// TIA Portal V16 export
// export: Created 2021-10-20T17:33:50.8567444Z, ExportSetting WithDefaults, DisplayName Totally Integrated Automation Portal, DisplayVersion V16, DisplayName TIA Portal Version Control Interface, DisplayVersion V16, DisplayName TIA Portal Openness, DisplayVersion V16, DisplayName TIA Portal Teamcenter Gateway, DisplayVersion V16, DisplayName SINAMICS Startdrive Advanced, DisplayVersion V16, DisplayName SINAMICS Startdrive G130, G150, S120, S150, SINAMICS MV, S210, DisplayVersion V16, DisplayName SINAMICS Startdrive G110M, G120, G120C, G120D, G120P, DisplayVersion V16, DisplayName STEP 7 Professional, DisplayVersion V16, DisplayName STEP 7 Safety, DisplayVersion V16, DisplayName WinCC Advanced, DisplayVersion V16
FUNCTION_BLOCK "Chillgard"   // FB2, LAD
TITLE = Chillgard analog communications
{ S7_Optimized_Access := 'TRUE' }
VERSION : 0.1
// Currently the Chillgard is only sensing 410A refrigerant.  More gas profiles may be added later.
// 
// Chillgard 5000 measures Rooms 16 & 19 - Indoor room, Indoor unit, Outdoor room, and Outdoor unit
// stored: AutoNumber true, IsIECCheckEnabled false, IsRetainMemResEnabled false, MemoryReserve 100, SetENOAutomatically false, UDAEnableTagReadback false
   VAR_TEMP   // added for the SCL form of the ladder/FBD networks
      _w1 : Bool;
      _w2 : Bool;
      _w3 : Bool;
      _w4 : Bool;
   END_VAR
BEGIN

REGION Network 1: Read and scale analog input values
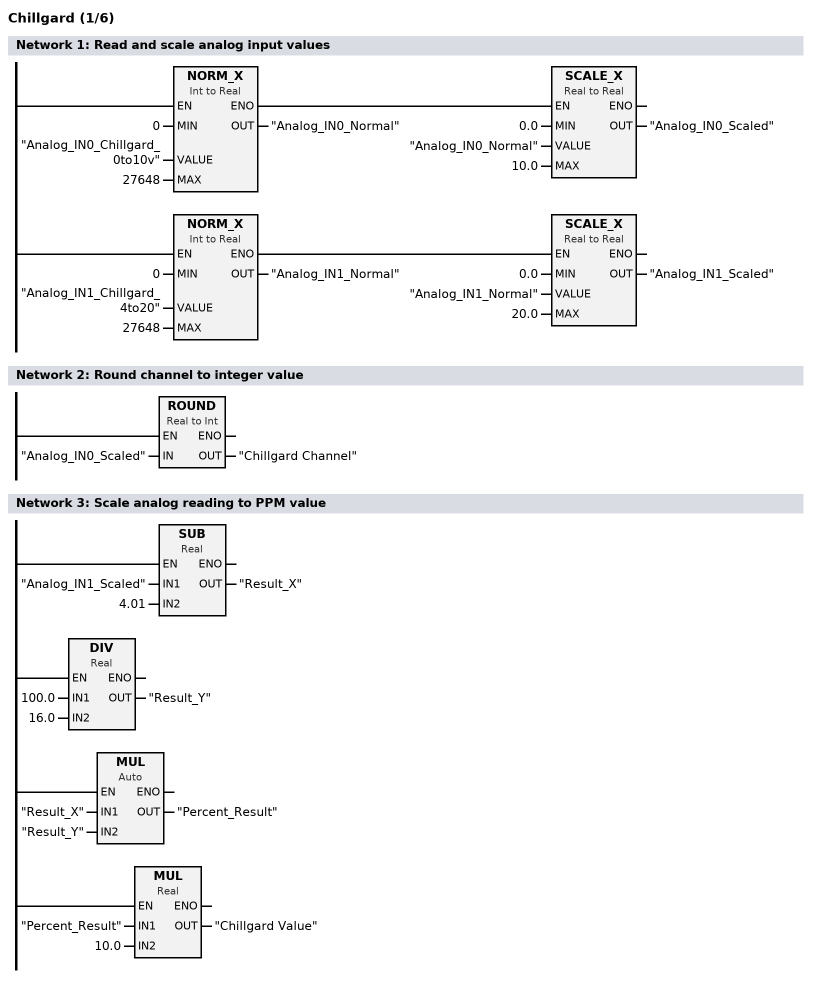
   RUNG wire#powerrail
      { S7_Templates := "[SrcType := Int, DestType := Real]" } Normalize(min := 0, value := "Analog_IN0_Chillgard_0to10v", max := 27648, out => "Analog_IN0_Normal")
      { S7_Templates := "[SrcType := Real, DestType := Real]" } Scale(min := 0.0, value := "Analog_IN0_Normal", max := 10.0, out => "Analog_IN0_Scaled")
   END_RUNG
   RUNG wire#powerrail
      { S7_Templates := "[SrcType := Int, DestType := Real]" } Normalize(min := 0, value := "Analog_IN1_Chillgard_4to20", max := 27648, out => "Analog_IN1_Normal")
      { S7_Templates := "[SrcType := Real, DestType := Real]" } Scale(min := 0.0, value := "Analog_IN1_Normal", max := 20.0, out => "Analog_IN1_Scaled")
   END_RUNG
   // the same network as SCL:
   "Analog_IN0_Normal" := NORM_X(MIN := 0, VALUE := "Analog_IN0_Chillgard_0to10v", MAX := 27648);
   "Analog_IN0_Scaled" := SCALE_X(MIN := 0.0, VALUE := "Analog_IN0_Normal", MAX := 10.0);
   "Analog_IN1_Normal" := NORM_X(MIN := 0, VALUE := "Analog_IN1_Chillgard_4to20", MAX := 27648);
   "Analog_IN1_Scaled" := SCALE_X(MIN := 0.0, VALUE := "Analog_IN1_Normal", MAX := 20.0);
END_REGION

REGION Network 2: Round channel to integer value
   RUNG wire#powerrail
      { S7_Templates := "[SrcType := Real, DestType := Int]" } Round(in := "Analog_IN0_Scaled", out => "Chillgard Channel")
   END_RUNG
   // the same network as SCL:
   "Chillgard Channel" := ROUND("Analog_IN0_Scaled");
END_REGION

REGION Network 3: Scale analog reading to PPM value
   RUNG wire#powerrail
      { S7_Templates := "SrcType := Real" } Sub(in1 := "Analog_IN1_Scaled", in2 := 4.01, out => "Result_X")
   END_RUNG
   RUNG wire#powerrail
      { S7_Templates := "SrcType := Real" } Div(in1 := 100.0, in2 := 16.0, out => "Result_Y")
   END_RUNG
   RUNG wire#powerrail
      Mul(in1 := "Result_X", in2 := "Result_Y", out => "Percent_Result")
   END_RUNG
   RUNG wire#powerrail
      { S7_Templates := "SrcType := Real" } Mul(in1 := "Percent_Result", in2 := 10.0, out => "Chillgard Value")
   END_RUNG
   // the same network as SCL:
   "Result_X" := "Analog_IN1_Scaled" - 4.01;
   "Result_Y" := 100.0 / 16.0;
   "Percent_Result" := "Result_X" * "Result_Y";
   "Chillgard Value" := "Percent_Result" * 10.0;
END_REGION

REGION Network 4: Assign values to proper channels - Room 4
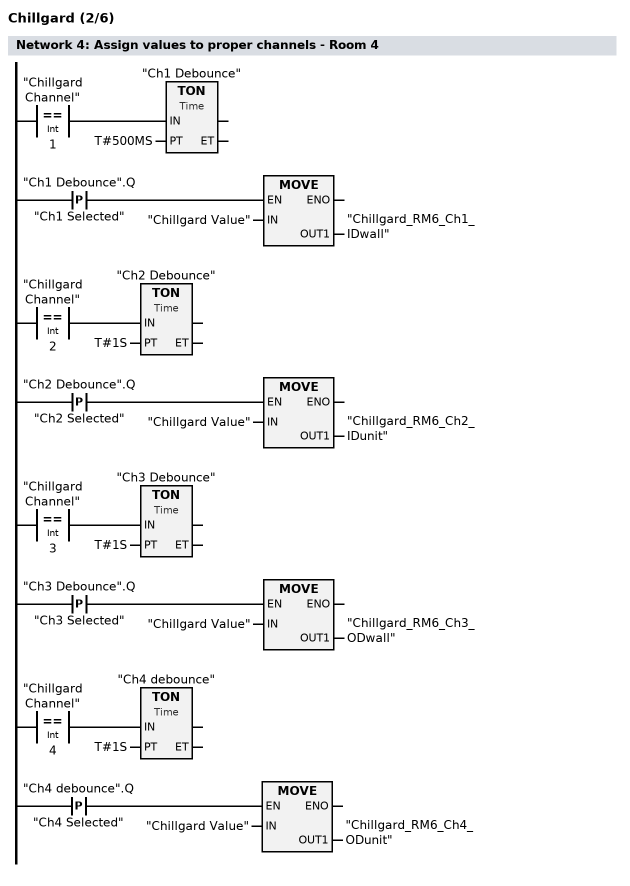
   RUNG wire#powerrail
      { S7_Templates := "SrcType := Int" } EQ_Contact(in1 := "Chillgard Channel", in2 := 1)
      { S7_Templates := "time_type := Time" } "Ch1 Debounce".TON(pt := T#500MS, et =>)
   END_RUNG
   RUNG wire#powerrail
      P_Contact(operand := "Ch1 Debounce".Q, bit := "Ch1 Selected")
      Move(in := "Chillgard Value", out1 => "Chillgard_RM6_Ch1_IDwall")
   END_RUNG
   RUNG wire#powerrail
      { S7_Templates := "SrcType := Int" } EQ_Contact(in1 := "Chillgard Channel", in2 := 2)
      { S7_Templates := "time_type := Time" } "Ch2 Debounce".TON(pt := T#1S, et =>)
   END_RUNG
   RUNG wire#powerrail
      P_Contact(operand := "Ch2 Debounce".Q, bit := "Ch2 Selected")
      Move(in := "Chillgard Value", out1 => "Chillgard_RM6_Ch2_IDunit")
   END_RUNG
   RUNG wire#powerrail
      { S7_Templates := "SrcType := Int" } EQ_Contact(in1 := "Chillgard Channel", in2 := 3)
      { S7_Templates := "time_type := Time" } "Ch3 Debounce".TON(pt := T#1S, et =>)
   END_RUNG
   RUNG wire#powerrail
      P_Contact(operand := "Ch3 Debounce".Q, bit := "Ch3 Selected")
      Move(in := "Chillgard Value", out1 => "Chillgard_RM6_Ch3_ODwall")
   END_RUNG
   RUNG wire#powerrail
      { S7_Templates := "SrcType := Int" } EQ_Contact(in1 := "Chillgard Channel", in2 := 4)
      { S7_Templates := "time_type := Time" } "Ch4 debounce".TON(pt := T#1S, et =>)
   END_RUNG
   RUNG wire#powerrail
      P_Contact(operand := "Ch4 debounce".Q, bit := "Ch4 Selected")
      Move(in := "Chillgard Value", out1 => "Chillgard_RM6_Ch4_ODunit")
   END_RUNG
   // the same network as SCL:
   "Ch1 Debounce".TON(IN := "Chillgard Channel" = 1, PT := T#500MS);
   #_w1 := "Ch1 Debounce".Q AND NOT "Ch1 Selected";   // rising edge of "Ch1 Debounce".Q
   "Ch1 Selected" := "Ch1 Debounce".Q;
   IF #_w1 THEN "Chillgard_RM6_Ch1_IDwall" := "Chillgard Value"; END_IF;
   "Ch2 Debounce".TON(IN := "Chillgard Channel" = 2, PT := T#1S);
   #_w2 := "Ch2 Debounce".Q AND NOT "Ch2 Selected";   // rising edge of "Ch2 Debounce".Q
   "Ch2 Selected" := "Ch2 Debounce".Q;
   IF #_w2 THEN "Chillgard_RM6_Ch2_IDunit" := "Chillgard Value"; END_IF;
   "Ch3 Debounce".TON(IN := "Chillgard Channel" = 3, PT := T#1S);
   #_w3 := "Ch3 Debounce".Q AND NOT "Ch3 Selected";   // rising edge of "Ch3 Debounce".Q
   "Ch3 Selected" := "Ch3 Debounce".Q;
   IF #_w3 THEN "Chillgard_RM6_Ch3_ODwall" := "Chillgard Value"; END_IF;
   "Ch4 debounce".TON(IN := "Chillgard Channel" = 4, PT := T#1S);
   #_w4 := "Ch4 debounce".Q AND NOT "Ch4 Selected";   // rising edge of "Ch4 debounce".Q
   "Ch4 Selected" := "Ch4 debounce".Q;
   IF #_w4 THEN "Chillgard_RM6_Ch4_ODunit" := "Chillgard Value"; END_IF;
END_REGION

REGION Network 5: Assign values to proper channels - Room 5
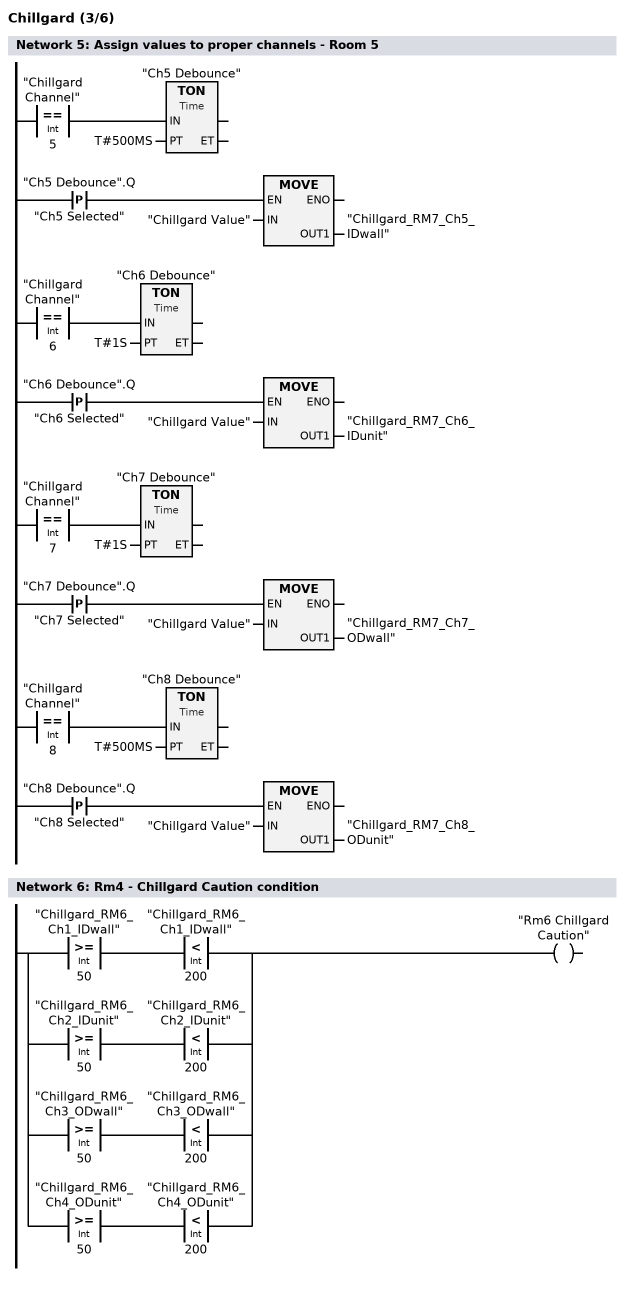
   RUNG wire#powerrail
      { S7_Templates := "SrcType := Int" } EQ_Contact(in1 := "Chillgard Channel", in2 := 5)
      { S7_Templates := "time_type := Time" } "Ch5 Debounce".TON(pt := T#500MS, et =>)
   END_RUNG
   RUNG wire#powerrail
      P_Contact(operand := "Ch5 Debounce".Q, bit := "Ch5 Selected")
      Move(in := "Chillgard Value", out1 => "Chillgard_RM7_Ch5_IDwall")
   END_RUNG
   RUNG wire#powerrail
      { S7_Templates := "SrcType := Int" } EQ_Contact(in1 := "Chillgard Channel", in2 := 6)
      { S7_Templates := "time_type := Time" } "Ch6 Debounce".TON(pt := T#1S, et =>)
   END_RUNG
   RUNG wire#powerrail
      P_Contact(operand := "Ch6 Debounce".Q, bit := "Ch6 Selected")
      Move(in := "Chillgard Value", out1 => "Chillgard_RM7_Ch6_IDunit")
   END_RUNG
   RUNG wire#powerrail
      { S7_Templates := "SrcType := Int" } EQ_Contact(in1 := "Chillgard Channel", in2 := 7)
      { S7_Templates := "time_type := Time" } "Ch7 Debounce".TON(pt := T#1S, et =>)
   END_RUNG
   RUNG wire#powerrail
      P_Contact(operand := "Ch7 Debounce".Q, bit := "Ch7 Selected")
      Move(in := "Chillgard Value", out1 => "Chillgard_RM7_Ch7_ODwall")
   END_RUNG
   RUNG wire#powerrail
      { S7_Templates := "SrcType := Int" } EQ_Contact(in1 := "Chillgard Channel", in2 := 8)
      { S7_Templates := "time_type := Time" } "Ch8 Debounce".TON(pt := T#500MS, et =>)
   END_RUNG
   RUNG wire#powerrail
      P_Contact(operand := "Ch8 Debounce".Q, bit := "Ch8 Selected")
      Move(in := "Chillgard Value", out1 => "Chillgard_RM7_Ch8_ODunit")
   END_RUNG
   // the same network as SCL:
   "Ch5 Debounce".TON(IN := "Chillgard Channel" = 5, PT := T#500MS);
   #_w1 := "Ch5 Debounce".Q AND NOT "Ch5 Selected";   // rising edge of "Ch5 Debounce".Q
   "Ch5 Selected" := "Ch5 Debounce".Q;
   IF #_w1 THEN "Chillgard_RM7_Ch5_IDwall" := "Chillgard Value"; END_IF;
   "Ch6 Debounce".TON(IN := "Chillgard Channel" = 6, PT := T#1S);
   #_w2 := "Ch6 Debounce".Q AND NOT "Ch6 Selected";   // rising edge of "Ch6 Debounce".Q
   "Ch6 Selected" := "Ch6 Debounce".Q;
   IF #_w2 THEN "Chillgard_RM7_Ch6_IDunit" := "Chillgard Value"; END_IF;
   "Ch7 Debounce".TON(IN := "Chillgard Channel" = 7, PT := T#1S);
   #_w3 := "Ch7 Debounce".Q AND NOT "Ch7 Selected";   // rising edge of "Ch7 Debounce".Q
   "Ch7 Selected" := "Ch7 Debounce".Q;
   IF #_w3 THEN "Chillgard_RM7_Ch7_ODwall" := "Chillgard Value"; END_IF;
   "Ch8 Debounce".TON(IN := "Chillgard Channel" = 8, PT := T#500MS);
   #_w4 := "Ch8 Debounce".Q AND NOT "Ch8 Selected";   // rising edge of "Ch8 Debounce".Q
   "Ch8 Selected" := "Ch8 Debounce".Q;
   IF #_w4 THEN "Chillgard_RM7_Ch8_ODunit" := "Chillgard Value"; END_IF;
END_REGION

REGION Network 6: Rm4 - Chillgard Caution condition
   RUNG wire#powerrail
      { S7_Templates := "SrcType := Int" } GE_Contact(in1 := "Chillgard_RM6_Ch1_IDwall", in2 := 50)
      { S7_Templates := "SrcType := Int" } LT_Contact(in1 := "Chillgard_RM6_Ch1_IDwall", in2 := 200)
      wire#w1
      Coil( "Rm6 Chillgard Caution" )
   END_RUNG
   RUNG wire#powerrail
      { S7_Templates := "SrcType := Int" } GE_Contact(in1 := "Chillgard_RM6_Ch2_IDunit", in2 := 50)
      { S7_Templates := "SrcType := Int" } LT_Contact(in1 := "Chillgard_RM6_Ch2_IDunit", in2 := 200)
   END_RUNG wire#w1
   RUNG wire#powerrail
      { S7_Templates := "SrcType := Int" } GE_Contact(in1 := "Chillgard_RM6_Ch3_ODwall", in2 := 50)
      { S7_Templates := "SrcType := Int" } LT_Contact(in1 := "Chillgard_RM6_Ch3_ODwall", in2 := 200)
   END_RUNG wire#w1
   RUNG wire#powerrail
      { S7_Templates := "SrcType := Int" } GE_Contact(in1 := "Chillgard_RM6_Ch4_ODunit", in2 := 50)
      { S7_Templates := "SrcType := Int" } LT_Contact(in1 := "Chillgard_RM6_Ch4_ODunit", in2 := 200)
   END_RUNG wire#w1
   // the same network as SCL:
   "Rm6 Chillgard Caution" := (("Chillgard_RM6_Ch1_IDwall" >= 50) AND ("Chillgard_RM6_Ch1_IDwall" < 200)) OR (("Chillgard_RM6_Ch2_IDunit" >= 50) AND ("Chillgard_RM6_Ch2_IDunit" < 200)) OR (("Chillgard_RM6_Ch3_ODwall" >= 50) AND ("Chillgard_RM6_Ch3_ODwall" < 200)) OR (("Chillgard_RM6_Ch4_ODunit" >= 50) AND ("Chillgard_RM6_Ch4_ODunit" < 200));
END_REGION

REGION Network 7: Rm4 - Chillgard Warning Condition
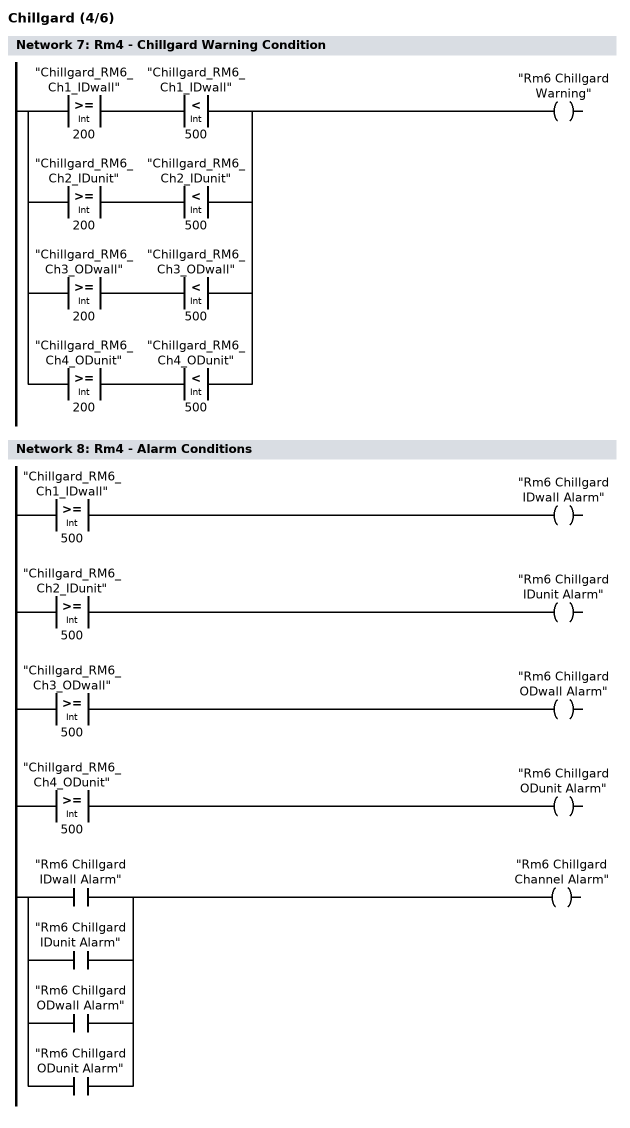
   RUNG wire#powerrail
      { S7_Templates := "SrcType := Int" } GE_Contact(in1 := "Chillgard_RM6_Ch1_IDwall", in2 := 200)
      { S7_Templates := "SrcType := Int" } LT_Contact(in1 := "Chillgard_RM6_Ch1_IDwall", in2 := 500)
      wire#w1
      Coil( "Rm6 Chillgard Warning" )
   END_RUNG
   RUNG wire#powerrail
      { S7_Templates := "SrcType := Int" } GE_Contact(in1 := "Chillgard_RM6_Ch2_IDunit", in2 := 200)
      { S7_Templates := "SrcType := Int" } LT_Contact(in1 := "Chillgard_RM6_Ch2_IDunit", in2 := 500)
   END_RUNG wire#w1
   RUNG wire#powerrail
      { S7_Templates := "SrcType := Int" } GE_Contact(in1 := "Chillgard_RM6_Ch3_ODwall", in2 := 200)
      { S7_Templates := "SrcType := Int" } LT_Contact(in1 := "Chillgard_RM6_Ch3_ODwall", in2 := 500)
   END_RUNG wire#w1
   RUNG wire#powerrail
      { S7_Templates := "SrcType := Int" } GE_Contact(in1 := "Chillgard_RM6_Ch4_ODunit", in2 := 200)
      { S7_Templates := "SrcType := Int" } LT_Contact(in1 := "Chillgard_RM6_Ch4_ODunit", in2 := 500)
   END_RUNG wire#w1
   // the same network as SCL:
   "Rm6 Chillgard Warning" := (("Chillgard_RM6_Ch1_IDwall" >= 200) AND ("Chillgard_RM6_Ch1_IDwall" < 500)) OR (("Chillgard_RM6_Ch2_IDunit" >= 200) AND ("Chillgard_RM6_Ch2_IDunit" < 500)) OR (("Chillgard_RM6_Ch3_ODwall" >= 200) AND ("Chillgard_RM6_Ch3_ODwall" < 500)) OR (("Chillgard_RM6_Ch4_ODunit" >= 200) AND ("Chillgard_RM6_Ch4_ODunit" < 500));
END_REGION

REGION Network 8: Rm4 - Alarm Conditions
   RUNG wire#powerrail
      { S7_Templates := "SrcType := Int" } GE_Contact(in1 := "Chillgard_RM6_Ch1_IDwall", in2 := 500)
      Coil( "Rm6 Chillgard IDwall Alarm" )
   END_RUNG
   RUNG wire#powerrail
      { S7_Templates := "SrcType := Int" } GE_Contact(in1 := "Chillgard_RM6_Ch2_IDunit", in2 := 500)
      Coil( "Rm6 Chillgard IDunit Alarm" )
   END_RUNG
   RUNG wire#powerrail
      { S7_Templates := "SrcType := Int" } GE_Contact(in1 := "Chillgard_RM6_Ch3_ODwall", in2 := 500)
      Coil( "Rm6 Chillgard ODwall Alarm" )
   END_RUNG
   RUNG wire#powerrail
      { S7_Templates := "SrcType := Int" } GE_Contact(in1 := "Chillgard_RM6_Ch4_ODunit", in2 := 500)
      Coil( "Rm6 Chillgard ODunit Alarm" )
   END_RUNG
   RUNG wire#powerrail
      Contact( "Rm6 Chillgard IDwall Alarm" )
      wire#w1
      Coil( "Rm6 Chillgard Channel Alarm" )
   END_RUNG
   RUNG wire#powerrail
      Contact( "Rm6 Chillgard IDunit Alarm" )
   END_RUNG wire#w1
   RUNG wire#powerrail
      Contact( "Rm6 Chillgard ODwall Alarm" )
   END_RUNG wire#w1
   RUNG wire#powerrail
      Contact( "Rm6 Chillgard ODunit Alarm" )
   END_RUNG wire#w1
   // the same network as SCL:
   "Rm6 Chillgard IDwall Alarm" := "Chillgard_RM6_Ch1_IDwall" >= 500;
   "Rm6 Chillgard IDunit Alarm" := "Chillgard_RM6_Ch2_IDunit" >= 500;
   "Rm6 Chillgard ODwall Alarm" := "Chillgard_RM6_Ch3_ODwall" >= 500;
   "Rm6 Chillgard ODunit Alarm" := "Chillgard_RM6_Ch4_ODunit" >= 500;
   "Rm6 Chillgard Channel Alarm" := "Rm6 Chillgard IDwall Alarm" OR "Rm6 Chillgard IDunit Alarm" OR "Rm6 Chillgard ODwall Alarm" OR "Rm6 Chillgard ODunit Alarm";
END_REGION

REGION Network 9: Rm5 - Chillgard Caution Condition
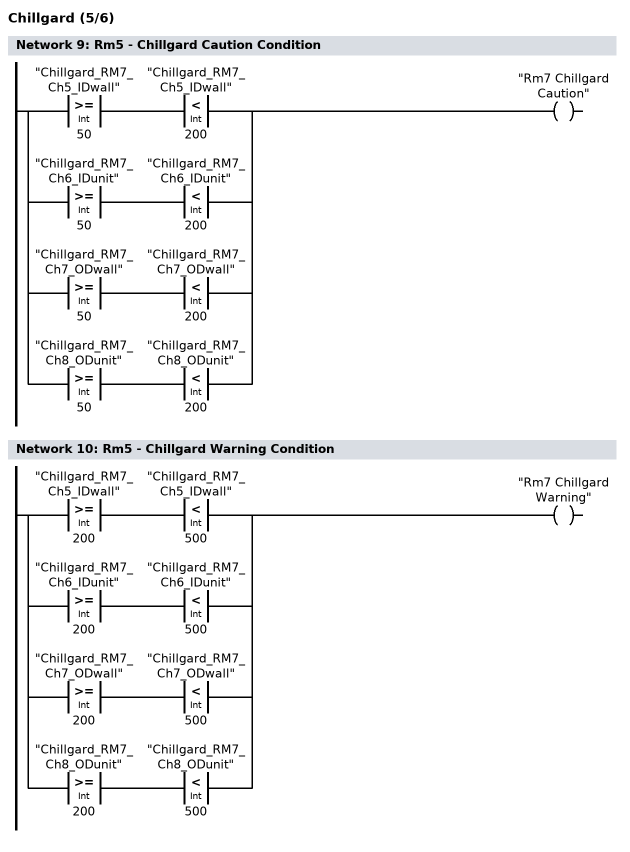
   RUNG wire#powerrail
      { S7_Templates := "SrcType := Int" } GE_Contact(in1 := "Chillgard_RM7_Ch5_IDwall", in2 := 50)
      { S7_Templates := "SrcType := Int" } LT_Contact(in1 := "Chillgard_RM7_Ch5_IDwall", in2 := 200)
      wire#w1
      Coil( "Rm7 Chillgard Caution" )
   END_RUNG
   RUNG wire#powerrail
      { S7_Templates := "SrcType := Int" } GE_Contact(in1 := "Chillgard_RM7_Ch6_IDunit", in2 := 50)
      { S7_Templates := "SrcType := Int" } LT_Contact(in1 := "Chillgard_RM7_Ch6_IDunit", in2 := 200)
   END_RUNG wire#w1
   RUNG wire#powerrail
      { S7_Templates := "SrcType := Int" } GE_Contact(in1 := "Chillgard_RM7_Ch7_ODwall", in2 := 50)
      { S7_Templates := "SrcType := Int" } LT_Contact(in1 := "Chillgard_RM7_Ch7_ODwall", in2 := 200)
   END_RUNG wire#w1
   RUNG wire#powerrail
      { S7_Templates := "SrcType := Int" } GE_Contact(in1 := "Chillgard_RM7_Ch8_ODunit", in2 := 50)
      { S7_Templates := "SrcType := Int" } LT_Contact(in1 := "Chillgard_RM7_Ch8_ODunit", in2 := 200)
   END_RUNG wire#w1
   // the same network as SCL:
   "Rm7 Chillgard Caution" := (("Chillgard_RM7_Ch5_IDwall" >= 50) AND ("Chillgard_RM7_Ch5_IDwall" < 200)) OR (("Chillgard_RM7_Ch6_IDunit" >= 50) AND ("Chillgard_RM7_Ch6_IDunit" < 200)) OR (("Chillgard_RM7_Ch7_ODwall" >= 50) AND ("Chillgard_RM7_Ch7_ODwall" < 200)) OR (("Chillgard_RM7_Ch8_ODunit" >= 50) AND ("Chillgard_RM7_Ch8_ODunit" < 200));
END_REGION

REGION Network 10: Rm5 - Chillgard Warning Condition
   RUNG wire#powerrail
      { S7_Templates := "SrcType := Int" } GE_Contact(in1 := "Chillgard_RM7_Ch5_IDwall", in2 := 200)
      { S7_Templates := "SrcType := Int" } LT_Contact(in1 := "Chillgard_RM7_Ch5_IDwall", in2 := 500)
      wire#w1
      Coil( "Rm7 Chillgard Warning" )
   END_RUNG
   RUNG wire#powerrail
      { S7_Templates := "SrcType := Int" } GE_Contact(in1 := "Chillgard_RM7_Ch6_IDunit", in2 := 200)
      { S7_Templates := "SrcType := Int" } LT_Contact(in1 := "Chillgard_RM7_Ch6_IDunit", in2 := 500)
   END_RUNG wire#w1
   RUNG wire#powerrail
      { S7_Templates := "SrcType := Int" } GE_Contact(in1 := "Chillgard_RM7_Ch7_ODwall", in2 := 200)
      { S7_Templates := "SrcType := Int" } LT_Contact(in1 := "Chillgard_RM7_Ch7_ODwall", in2 := 500)
   END_RUNG wire#w1
   RUNG wire#powerrail
      { S7_Templates := "SrcType := Int" } GE_Contact(in1 := "Chillgard_RM7_Ch8_ODunit", in2 := 200)
      { S7_Templates := "SrcType := Int" } LT_Contact(in1 := "Chillgard_RM7_Ch8_ODunit", in2 := 500)
   END_RUNG wire#w1
   // the same network as SCL:
   "Rm7 Chillgard Warning" := (("Chillgard_RM7_Ch5_IDwall" >= 200) AND ("Chillgard_RM7_Ch5_IDwall" < 500)) OR (("Chillgard_RM7_Ch6_IDunit" >= 200) AND ("Chillgard_RM7_Ch6_IDunit" < 500)) OR (("Chillgard_RM7_Ch7_ODwall" >= 200) AND ("Chillgard_RM7_Ch7_ODwall" < 500)) OR (("Chillgard_RM7_Ch8_ODunit" >= 200) AND ("Chillgard_RM7_Ch8_ODunit" < 500));
END_REGION

REGION Network 11: Rm5 - Chillgard Alarm Conditions
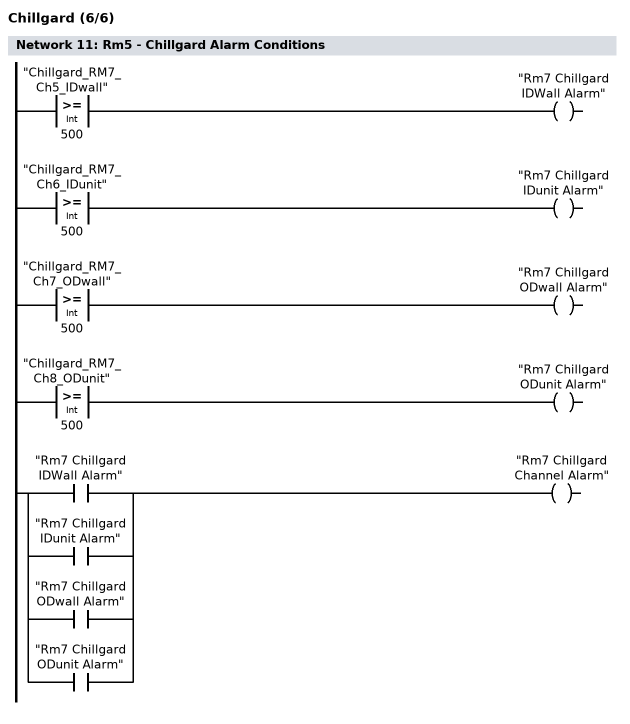
   RUNG wire#powerrail
      { S7_Templates := "SrcType := Int" } GE_Contact(in1 := "Chillgard_RM7_Ch5_IDwall", in2 := 500)
      Coil( "Rm7 Chillgard IDWall Alarm" )
   END_RUNG
   RUNG wire#powerrail
      { S7_Templates := "SrcType := Int" } GE_Contact(in1 := "Chillgard_RM7_Ch6_IDunit", in2 := 500)
      Coil( "Rm7 Chillgard IDunit Alarm" )
   END_RUNG
   RUNG wire#powerrail
      { S7_Templates := "SrcType := Int" } GE_Contact(in1 := "Chillgard_RM7_Ch7_ODwall", in2 := 500)
      Coil( "Rm7 Chillgard ODwall Alarm" )
   END_RUNG
   RUNG wire#powerrail
      { S7_Templates := "SrcType := Int" } GE_Contact(in1 := "Chillgard_RM7_Ch8_ODunit", in2 := 500)
      Coil( "Rm7 Chillgard ODunit Alarm" )
   END_RUNG
   RUNG wire#powerrail
      Contact( "Rm7 Chillgard IDWall Alarm" )
      wire#w1
      Coil( "Rm7 Chillgard Channel Alarm" )
   END_RUNG
   RUNG wire#powerrail
      Contact( "Rm7 Chillgard IDunit Alarm" )
   END_RUNG wire#w1
   RUNG wire#powerrail
      Contact( "Rm7 Chillgard ODwall Alarm" )
   END_RUNG wire#w1
   RUNG wire#powerrail
      Contact( "Rm7 Chillgard ODunit Alarm" )
   END_RUNG wire#w1
   // the same network as SCL:
   "Rm7 Chillgard IDWall Alarm" := "Chillgard_RM7_Ch5_IDwall" >= 500;
   "Rm7 Chillgard IDunit Alarm" := "Chillgard_RM7_Ch6_IDunit" >= 500;
   "Rm7 Chillgard ODwall Alarm" := "Chillgard_RM7_Ch7_ODwall" >= 500;
   "Rm7 Chillgard ODunit Alarm" := "Chillgard_RM7_Ch8_ODunit" >= 500;
   "Rm7 Chillgard Channel Alarm" := "Rm7 Chillgard IDWall Alarm" OR "Rm7 Chillgard IDunit Alarm" OR "Rm7 Chillgard ODwall Alarm" OR "Rm7 Chillgard ODunit Alarm";
END_REGION
END_FUNCTION_BLOCK
